TYPE (* ISOBUS UT scroll list operator controls (6 buttons + direct-position input field) *)
  (* Standard: 61499-2; Description: Copyright (c) 2026 Meisterschulen am Ostbahnhof This program and the accompanying materials are made available under the terms of the Eclipse Public License 2.0 which is available at https://www.eclipse.org/legal/epl-2.0/ SPDX-License-Identifier: EPL-2.0 *)
  (* Version 1.0, 2026-08-09, Franz Höpfinger, Meisterschulen am Ostbahnhof, initial API and implementation and/or initial documentation *)
  PACKAGE isobus::utils::scroll;
  IMPORT isobus::UT::Q::const::IDs;
  ScrollControls_S : STRUCT
    u16BtnTopId : UINT := IDs::ID_NULL; (* Object ID of the softkey/button that fires the TOP event *)
    u16BtnPageUpId : UINT := IDs::ID_NULL; (* Object ID of the softkey/button that fires the UP_UP event *)
    u16BtnUpId : UINT := IDs::ID_NULL; (* Object ID of the softkey/button that fires the UP event *)
    u16BtnDownId : UINT := IDs::ID_NULL; (* Object ID of the softkey/button that fires the DOWN event *)
    u16BtnPageDownId : UINT := IDs::ID_NULL; (* Object ID of the softkey/button that fires the DOWN_DOWN event *)
    u16BtnBottomId : UINT := IDs::ID_NULL; (* Object ID of the softkey/button that fires the BOTTOM event *)
    u16GotoInputId : UINT := IDs::ID_NULL; (* Object ID of the InputNumber field for direct row-position entry (drives the POS/GOTO event's SET_POS value) *)
  END_STRUCT;
END_TYPE
